(*
Registers component. Alternative function block: `Comp`.
*)
FUNCTION RegComp : Result
VAR_INPUT
	iComponent	: I_Component;
	iEntity		: I_Entity;
END_VAR
VAR
	_nResult	: Result;
END_VAR

RegComp := _RegComp(iEntity, iComponent);

END_FUNCTION

(* stored: Version 1.1.0.1
   POU RegComp: Id {9d5059a5-7ec0-4c08-8587-3adfec1dbc46}, SpecialFunc None *)
